TYPE TcoEvaluateMeasurementResults : 
STRUCT
    RisingPeaks : ARRAY[0..100] OF TcoEvaluateMeasurementDataItem;
    RisingPeaksFound : INT;
    FallingPeaks : ARRAY[0..100] OF TcoEvaluateMeasurementDataItem;
    FallingPeaksFound : INT;
    Triggers : ARRAY[0..100] OF TcoEvaluateMeasurementDataItem;
    TriggersFound : INT;
END_STRUCT
END_TYPE

(* stored: Version 1.1.0.1, ProductVersion 3.1.4024.10
   DUT TcoEvaluateMeasurementResults: Id {a0daa1d8-5432-0dff-2035-6c88435cf77d} *)
